{attribute 'qualified_only'}
VAR_GLOBAL
	
	DHR_RollingSchedule 	: ST_DHR_Rollingschedule_Entry;

END_VAR

(* stored: Version 1.1.0.1, ProductVersion 3.1.4024.2
   GVL GVL_Visu: Id {55d75e8c-4410-40ad-8aa3-92c4e7997893} *)
